INTERFACE I_State EXTENDS I_Base

METHOD Executing : BOOL;
END_METHOD

METHOD Inactive
VAR_INPUT
END_VAR
END_METHOD

END_INTERFACE

(* stored: Version 1.1.0.1, ProductVersion 3.1.4026.18
   Itf I_State: Id {41b16221-ed23-481e-917f-ecd9f8eb4019}
   Method Executing: Id {25260be4-d9ad-42ad-ba45-7deccc8e3716}
   Method Inactive: Id {8ded77ff-6605-4d71-9ab3-b5ce2ff39e5e} *)
